# B&R Automation Studio project LabRab1
Automation Studio 4.9

## Configuration Config1

CPU 4PP065.0351-P74, AutomationRuntime B4.91, Build 4.1.2, Vc V4.72.3

### Task classes (Cpu.sw)
```
Cyclic#1:
  Program <- Program.prg
Binaries: udbdef, FWRules, TCData, sysconf, Role, User, iomap, ashwd, asfw, arconfig, ashwac
Libraries: MotorCntrl
```

### Hardware
```
4PP065_0351_P74 : 4PP065.0351-P74 v1.0.4.0
  Connector IF5:
    ActivateDevice = 1
  ConfigurationID = Lab1_Config1
  Simulation = 1
  FileDevice1
  FileDeviceName1 = USER
  FileDevicePath1 = USER_PATH
  KeyMappingFile = VC\4PP065_0351_P74.dis
```

## Logical view

### Program Logical/Program (ANSIC)

#### Variables.var
```iecst
VAR
	fb_regulator : FB_Regulator;
	fb_motor : FB_Motor;
	speed : REAL;
	Enable : BOOL;
	fb_motor1 : FB_Motor1;
	t : REAL;
END_VAR
```

#### Cyclic.c
```c
#include <bur/plctypes.h>

#ifdef _DEFAULT_INCLUDES
	#include <AsDefault.h>
#endif

void _CYCLIC ProgramCyclic(void)
{
	if (Enable == 1)
	{
		speed = 100;
	}
	if (Enable == 0)
	{
		speed = 0;
	}
	t = t + 0.01;
	fb_regulator.e = speed - fb_motor.w;
	FB_Regulator(&fb_regulator);
	fb_motor.u = fb_regulator.u;
	FB_Motor(&fb_motor);

	FB_Motor1(&fb_motor1);
	fb_motor1.u = speed - fb_motor1.w;

	if ((t > 2)){
		Enable = !Enable;
		t = 0;
	}
}
```

#### Init.c
```c
#include <bur/plctypes.h>

#ifdef _DEFAULT_INCLUDES
	#include <AsDefault.h>
#endif

void _INIT ProgramInit(void)
{
	t = 0;
	fb_regulator.k_i = 0.16;
	fb_regulator.k_p = 0.0064;
	fb_motor.dt = 0.01;
	fb_motor.Tm = 0.004;
	fb_motor.ke = 0.0002;
	fb_regulator.dt = 0.01;
	fb_regulator.e = 0;
	fb_regulator.max_abs_value = 300;
	fb_motor1.u = 0;
	fb_motor1.dt = 0.01;
	fb_motor1.Tm = 0.01;
	fb_motor1.ke = 0.2;
	Enable  = 1;
}
```

### Library Logical/MotorCntrl (ANSIC)

#### MotorCntrl.fun - Exported functions and function blocks
```iecst
{REDUND_ERROR} FUNCTION_BLOCK FB_Integrator (*TODO: Add your comment here*) (*$GROUP=User,$CAT=User,$GROUPICON=User.png,$CATICON=User.png*)
	VAR_INPUT
		in : {REDUND_UNREPLICABLE} REAL;
	END_VAR
	VAR_OUTPUT
		out : {REDUND_UNREPLICABLE} REAL;
	END_VAR
	VAR
		dt : {REDUND_UNREPLICABLE} REAL;
		oldval : REAL;
	END_VAR
END_FUNCTION_BLOCK

{REDUND_ERROR} FUNCTION_BLOCK FB_Motor (*TODO: Add your comment here*) (*$GROUP=User,$CAT=User,$GROUPICON=User.png,$CATICON=User.png*)
	VAR_INPUT
		u : {REDUND_UNREPLICABLE} REAL;
		Tm : REAL;
	END_VAR
	VAR_OUTPUT
		w : {REDUND_UNREPLICABLE} REAL;
		phi : {REDUND_UNREPLICABLE} REAL;
	END_VAR
	VAR
		integrator1 : FB_Integrator;
		integrator : {REDUND_UNREPLICABLE} FB_Integrator;
		ke : {REDUND_UNREPLICABLE} REAL;
		dt : {REDUND_UNREPLICABLE} REAL;
	END_VAR
END_FUNCTION_BLOCK

{REDUND_ERROR} FUNCTION_BLOCK FB_Regulator (*TODO: Add your comment here*) (*$GROUP=User,$CAT=User,$GROUPICON=User.png,$CATICON=User.png*)
	VAR
		e : REAL;
		u : REAL;
		k_p : {REDUND_UNREPLICABLE} REAL;
		k_i : {REDUND_UNREPLICABLE} REAL;
		integrator : {REDUND_UNREPLICABLE} FB_Integrator;
		iyOld : {REDUND_UNREPLICABLE} REAL;
		max_abs_value : {REDUND_UNREPLICABLE} REAL;
		dt : {REDUND_UNREPLICABLE} REAL;
	END_VAR
END_FUNCTION_BLOCK

{REDUND_ERROR} {REDUND_UNREPLICABLE} FUNCTION_BLOCK FB_Motor1 (*TODO: Add your comment here*) (*$GROUP=User,$CAT=User,$GROUPICON=User.png,$CATICON=User.png*)
	VAR_INPUT
		u : {REDUND_UNREPLICABLE} REAL;
		Tm : {REDUND_UNREPLICABLE} REAL;
	END_VAR
	VAR_OUTPUT
		w : {REDUND_UNREPLICABLE} REAL;
		phi : {REDUND_UNREPLICABLE} REAL;
	END_VAR
	VAR
		ke : {REDUND_UNREPLICABLE} REAL;
		integrator : {REDUND_UNREPLICABLE} FB_Integrator;
		integrator1 : {REDUND_UNREPLICABLE} FB_Integrator;
		dt : {REDUND_UNREPLICABLE} REAL;
	END_VAR
END_FUNCTION_BLOCK
```

#### FB_Integrator.c
```c
#include <bur/plctypes.h>
#ifdef __cplusplus
	extern "C"
	{
#endif
	#include "MotorCntrl.h"
#ifdef __cplusplus
	};
#endif
/* TODO: Add your comment here */
void FB_Integrator(struct FB_Integrator* inst)
{
	inst->out = inst->oldval + ((inst->in) * inst->dt);
	inst->oldval = inst->out;
}
```

#### FB_Motor.c
```c
#include <bur/plctypes.h>
#ifdef __cplusplus
	extern "C"
	{
#endif
	#include "MotorCntrl.h"
#ifdef __cplusplus
	};
#endif
/* TODO: Add your comment here */
void FB_Motor(struct FB_Motor* inst)
{
	REAL temp;
	temp = inst->u / inst->ke;
	temp = temp - inst->w;
	temp = temp * inst->dt / inst->Tm;
	inst->integrator.in = temp;
	inst->integrator.dt = inst->dt;
	inst->integrator1.dt = inst->dt;
	FB_Integrator(&inst->integrator);
	temp = inst->integrator.out;
	inst->w = temp;
	temp = inst->w;
	inst->integrator1.in = temp;
	FB_Integrator(&inst->integrator1);
	inst->phi = inst->integrator1.out;
}
```

#### FB_Regulator.c
```c
#include <bur/plctypes.h>
#ifdef __cplusplus
	extern "C"
	{
#endif
	#include "MotorCntrl.h"
#ifdef __cplusplus
	};
#endif
/* TODO: Add your comment here */
void FB_Regulator(struct FB_Regulator* inst)
{
	REAL temp;
	temp = inst->e * inst->k_i * inst->dt;
	temp+=inst->iyOld;
	inst->integrator.in = temp;
	inst->integrator.dt = inst->dt;
	FB_Integrator(&inst->integrator);

	if (inst->e * inst->k_p > inst->max_abs_value)
	{
		temp = inst->integrator.out + inst->max_abs_value;
	}
	if (inst->e * inst->k_p < inst->max_abs_value)
	{
		temp = inst->integrator.out + inst->e * inst->k_p;
	}
	if (temp > inst->max_abs_value)
	{
		inst->u = inst->max_abs_value;
		inst->iyOld = temp - inst->max_abs_value;
	}
	else
	{
		inst->u = temp;
		inst->iyOld = 0;
	}

}
```

#### FB_Motor1.c
```c
#include <bur/plctypes.h>
#ifdef __cplusplus
	extern "C"
	{
#endif
	#include "MotorCntrl.h"
#ifdef __cplusplus
	};
#endif
/* TODO: Add your comment here */
void FB_Motor1(struct FB_Motor1* inst)
{
	REAL temp;
	temp = inst->u / inst->ke;
	temp = temp - inst->w;
	temp = temp * inst->dt / inst->Tm;
	inst->integrator.in = temp;
	inst->integrator.dt = inst->dt;
	inst->integrator1.dt = inst->dt;
	FB_Integrator(&inst->integrator);
	temp = inst->integrator.out;
	inst->w = temp;
	temp = inst->w;
	inst->integrator1.in = temp;
	FB_Integrator(&inst->integrator1);
	inst->phi = inst->integrator1.out;
}
```

Listed in the project but not available here: Logical/Global.typ, Logical/Global.var, Logical/Libraries, Logical/MotorCntrl/Types.typ, Logical/MotorCntrl/Constants.var
